// TIA Portal V17 export
// export: Created 2023-12-22T15:03:02.8695906Z, ExportSetting WithDefaults, DisplayName Totally Integrated Automation Portal, DisplayVersion V17, DisplayName TIA Portal Openness, DisplayVersion V17, DisplayName TIA Portal Version Control Interface, DisplayVersion V17, DisplayName STEP 7 Professional, DisplayVersion V17, DisplayName STEP 7 Safety, DisplayVersion V17, DisplayName WinCC Advanced, DisplayVersion V17
DATA_BLOCK "LE_Final_DB"   // DB308
VERSION : 0.1
// stored: AutoNumber false, DBAccessibleFromOPCUA true, DBAccessibleFromWebserver true, InstanceOfName AI_ex, InstanceOfType FB
"AI_ex"
   // VAR_OUTPUT
   //    S_Alarm : Bool;
   // END_VAR
   // VAR_IN_OUT
   //    Signal : Int;
   //    Result : Real;
   // END_VAR
   // VAR RETAIN
   //    CMD : "CMD";
   //    Mode : Int;
   //    Status : Int;
   //    Use : Struct
   //       RTD { S7_SetPoint := 'True'} : Bool;
   //       Filter { S7_SetPoint := 'True'} : Bool;
   //       Inverse { S7_SetPoint := 'True'} : Bool;
   //       Indirect { S7_SetPoint := 'True'} : Bool;
   //       Status { S7_SetPoint := 'True'} : Bool;
   //       Light { S7_SetPoint := 'True'} : Bool;
   //       Lim_Low { S7_SetPoint := 'True'} : Bool;
   //       Lim_High { S7_SetPoint := 'True'} : Bool;
   //       Communication { S7_SetPoint := 'True'} : Bool;
   //    END_STRUCT;
   //    VmA : Real;
   //    RTD_c { S7_SetPoint := 'True'} : Real;
   //    Calibration { S7_SetPoint := 'True'} : Real;
   //    Converter { S7_SetPoint := 'True'} : "Converter_LAD";
   //    SP : Struct
   //       NC { S7_SetPoint := 'True'} : Real;
   //       SC { S7_SetPoint := 'True'} : Real;
   //       HH { S7_SetPoint := 'True'} : Real;
   //       H { S7_SetPoint := 'True'} : Real;
   //       L { S7_SetPoint := 'True'} : Real;
   //       LL { S7_SetPoint := 'True'} : Real;
   //    END_STRUCT;
   //    Tx { S7_SetPoint := 'True'} : Array[0..5] of "Time_R";
   //    Alarm : Struct
   //       ST : Bool;
   //       HH : Bool;
   //       H : Bool;
   //       L : Bool;
   //       LL : Bool;
   //       NC : Bool;
   //       SC : Bool;
   //    END_STRUCT;
   //    Alarms : Word;
   //    Events : Word;
   //    pos : Array[0..15] of Bool;
   //    Input_Type { S7_SetPoint := 'True'} : Int;
   //    CodeID { S7_SetPoint := 'True'} : Int;
   //    "Type" { S7_SetPoint := 'True'} : Int;
   //    ADDR { S7_SetPoint := 'True'} : Int;
   //    Filter_SP { S7_SetPoint := 'True'} : Int;
   //    "Name" { S7_SetPoint := 'True'} : String[5];
   //    Filter_DB : "Filter";
   //    Time_DTL { S7_SetPoint := 'True'} : DTL;
   // END_VAR
BEGIN
END_DATA_BLOCK
